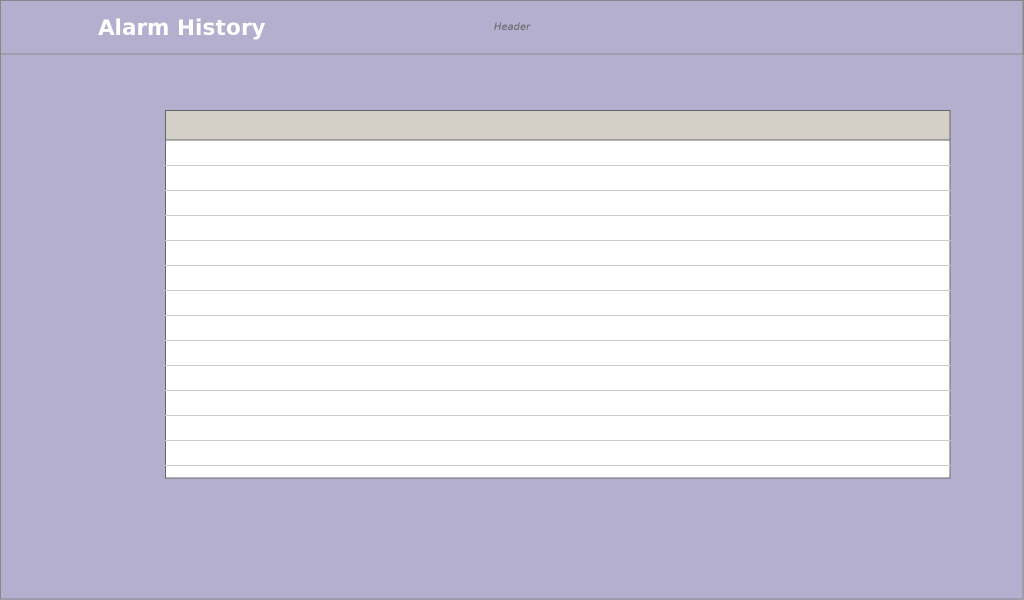
VISUALIZATION AlarmHistory  // 1024x600
    Frame (0,-1 1024x55)
        shows Header()
    Label (95,15 250x25), "Alarm History"
    Table (165,110 785x368), data array: status_Gvl.arAlarmHistory
        p3854506369: status_Gvl.arAlarmHistory[INDEX].Status
        p1892666644: status_Gvl.arAlarmHistory[INDEX].ErrorID
        p338671338: status_Gvl.arAlarmHistory[INDEX].ErrorMsg
        p2170511999: status_Gvl.arAlarmHistory[INDEX].TimeStop
        p511219082: Error ID
        p1755163831: Error Message
        p4092479075: Time Stop
END_VISUALIZATION

(* stored: Version 1.1.0.1, ProductVersion 3.1.4024.12
   Visu AlarmHistory: Id {d7adcfc8-d8bc-400d-8aac-3dbc8487f019} *)
